TYPE ARMType :
(
	ARMType_Default := 0, //常规的ARM
	ARMType_SinSun := 1, // 新松
	ARMType_Other := 2 // 蝶阀
)UINT;
END_TYPE

(* stored: Version 1.1.0.1, ProductVersion 3.1.4024.4
   DUT ARMType: Id {f40cc52a-a261-486c-a225-a6a372e0336f} *)
